{attribute addProperty BoxType "EL6001-0000-0020"}
{attribute addProperty Id "COM_InputsAT %I*COM_Inputs_F2FBC98A30COM_OutputsAT %Q*COM_Outputs_42B38F1527WcStateAT %I*WcState_9091E0EB2InfoDataAT %I*InfoData_32EB74EA10"}
{attribute addProperty CRC "2344280932"}
{attribute addProperty SizeInBites "552"}
{attribute addProperty SizeInBytes "69"}
TYPE EL6001_8BBAE364 :
STRUCT
	{attribute addProperty Name "COM_Inputs"}
	COM_Inputs : COM_Inputs_F2FBC98A;
	{attribute addProperty Name "COM_Outputs"}
	COM_Outputs : COM_Outputs_42B38F15;
	{attribute addProperty Name "WcState"}
	WcState : WcState_9091E0EB;
	{attribute addProperty Name "InfoData"}
	InfoData : InfoData_32EB74EA;
END_STRUCT
END_TYPE

(* stored: Version 1.2.0.0, ProductVersion 3.1.4024.9
   DUT EL6001_8BBAE364: Id {f2f18993-9ddd-4733-aa83-a7d3a23a022e} *)
